FUNCTION_BLOCK SimpleTestType2
  (* Version 1.0, 2008-12-19, Goran Cengic, Chalmers *)
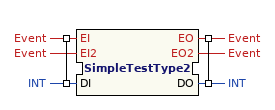
  EVENT_INPUT
    EI WITH DI;
    EI2;
  END_EVENT
  EVENT_OUTPUT
    EO WITH DO;
    EO2;
  END_EVENT
  VAR_INPUT
    DI : INT;
  END_VAR
  VAR_OUTPUT
    DO : INT;
  END_VAR
  VAR
    invoked : INT;
  END_VAR
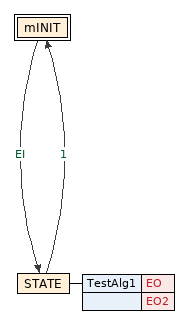
  EC_STATES
    mINIT;
    STATE : TestAlg1 -> EO, -> EO2;
  END_STATES
  EC_TRANSITIONS
    mINIT TO STATE := EI;
    STATE TO mINIT := 1;
  END_TRANSITIONS
  ALGORITHM TestAlg1 IN Java:
invoked++;
	DO = DI + 1;
	System.out.println("TestAlg:invoked: " + invoked + " times.");
	System.out.println("TestAlg: DO: " + DO + ".");
  END_ALGORITHM
END_FUNCTION_BLOCK
